FUNCTION_BLOCK LED_HMI (* 4-LED output emulator *)
  (* Standard: 61499 *)
  (* Version 0.1, 2008-06-04, JHC, Holobloc Inc, Updated DOCTYPE. *)
  (* Version 0.0, 2001-02-21, JHC, Rockwell Automation *)
  (* Compiler header: package fb.rt.ita; import fb.rt.hmi.*; *)
  (* Compiler Java IBM VisualAge 3.0 *)
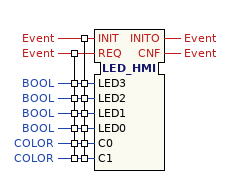
  EVENT_INPUT
    INIT WITH LED3, LED2, LED1, LED0, C0, C1; (* Initialization Request *)
    REQ WITH LED3, LED2, LED1, LED0, C0, C1; (* Display Request *)
  END_EVENT
  EVENT_OUTPUT
    INITO; (* Initialization Confirm *)
    CNF; (* Execution Confirmation *)
  END_EVENT
  VAR_INPUT
    LED3 : BOOL; (* MSB *)
    LED2 : BOOL;
    LED1 : BOOL;
    LED0 : BOOL; (* LSB *)
    C0 : COLOR := COLOR#white; (* OFF color *)
    C1 : COLOR := COLOR#orange; (* ON color *)
  END_VAR
  FBS
    OUT3 : OUT_BOOL;
    OUT2 : OUT_BOOL;
    OUT1 : OUT_BOOL;
    OUT0 : OUT_BOOL;
  END_FBS
  EVENT_CONNECTIONS
    INIT TO OUT3.INIT;
    OUT3.INITO TO OUT2.INIT;
    OUT2.INITO TO OUT1.INIT;
    OUT1.INITO TO OUT0.INIT;
    OUT0.INITO TO INITO;
    REQ TO OUT3.REQ;
    OUT3.CNF TO OUT2.REQ;
    OUT2.CNF TO OUT1.REQ;
    OUT1.CNF TO OUT0.REQ;
    OUT0.CNF TO CNF;
  END_CONNECTIONS
  DATA_CONNECTIONS
    1 TO OUT3.QI;
    1 TO OUT2.QI;
    1 TO OUT1.QI;
    1 TO OUT0.QI;
    "LED3" TO OUT3.LABEL;
    "LED2" TO OUT2.LABEL;
    "LED1" TO OUT1.LABEL;
    "LED0" TO OUT0.LABEL;
    LED3 TO OUT3.IN;
    LED2 TO OUT2.IN;
    LED1 TO OUT1.IN;
    LED0 TO OUT0.IN;
    C0 TO OUT3.C0;
    C0 TO OUT2.C0;
    C0 TO OUT1.C0;
    C0 TO OUT0.C0;
    C1 TO OUT3.C1;
    C1 TO OUT2.C1;
    C1 TO OUT1.C1;
    C1 TO OUT0.C1;
  END_CONNECTIONS
END_FUNCTION_BLOCK
